FUNCTION_BLOCK F_BAND_B (* Basic Function Block Type *)
  (* Standard: 61499-2; Classification: Control Modules; Description: BAND_B hides at the input areas 0..255 the areas 0..B and 255-B.. 255, in this areas the output is 0 respectively 255. *)
  (* Version 0.0, 2011-08-23, 4DIAC-IDE, 4DIAC-Consortium *)
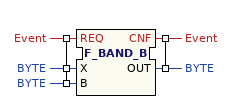
  EVENT_INPUT
    REQ WITH B, X; (* Normal Execution Request *)
  END_EVENT
  EVENT_OUTPUT
    CNF WITH OUT; (* Execution Confirmation *)
  END_EVENT
  VAR_INPUT
    X : BYTE; (* input value *)
    B : BYTE; (* limit area *)
  END_VAR
  VAR_OUTPUT
    OUT : BYTE; (* output value *)
  END_VAR
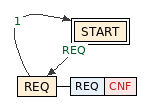
  EC_STATES
    START; (* Initial State *)
    REQ : REQ -> CNF; (* Normal execution *)
  END_STATES
  EC_TRANSITIONS
    START TO REQ := REQ;
    REQ TO START := 1;
  END_TRANSITIONS
  ALGORITHM REQ IN ST: (* Normally executed algorithm *)
IF X < B THEN
	OUT := 0;
ELSIF X > 255-B THEN
	OUT := 255;
ELSE
	OUT := X;
END_IF;
  END_ALGORITHM
END_FUNCTION_BLOCK
